FUNCTION_BLOCK PUBLIC FB_Logger
VAR
	ipLogger : ILogger;
END_VAR

METHOD FB_init : BOOL
VAR_INPUT
	bInitRetains       : BOOL; // if TRUE, the retain variables are initialized (warm start / cold start)
	bInCopyCode        : BOOL;  // if TRUE, the instance afterwards gets moved into the copy code (online change)
	refLoggerFactory   : REFERENCE TO FB_AbstractLoggerFactory;
END_VAR
IF (__ISVALIDREF(refLoggerFactory)) THEN
	ipLogger := refLoggerFactory.GetLogger();
ELSE
	ipLogger := 0;
END_IF
END_METHOD

METHOD PUBLIC Write : STRING
VAR_INPUT
	sMsg 		 : STRING;
END_VAR
Write := 'Error';
IF (ipLogger <> 0) THEN
	Write := ipLogger.Write(sMsg);
END_IF
END_METHOD

END_FUNCTION_BLOCK

(* stored: Version 1.1.0.1, ProductVersion 3.1.4022.18
   POU FB_Logger: Id {f01e87a0-60ff-4302-b8a9-762e186f392e}, SpecialFunc None
   Method FB_init: Id {7a98a545-7471-4e19-b87c-8a5d5190f2dc}
   Method Write: Id {34777f0c-26fa-45cc-9bc6-6bb5d033ffcd} *)
